// TIA Portal V18 export
VAR_GLOBAL   // PLC tag table "04_0 Costanti tipo attuatore"
END_VAR
VAR_GLOBAL CONSTANT   // user constants
   EV : Int := 1;
   MOT_POS : Int := 2;
   HMC : Int := 3;
   CNC : Int := 4;
   MOT_VEL : Int := 5;
   MOT_AA : Int := 6;
END_VAR
